// TIA Portal V20 export
// export: Created 2026-04-11T06:02:30.246913Z, ExportSetting WithDefaults, DisplayName Totally Integrated Automation Portal, DisplayVersion V20, DisplayName TIA Portal Openness, DisplayVersion V20, DisplayName TIA Portal Version Control Interface, DisplayVersion V20, DisplayName STEP 7 Professional, DisplayVersion V20, DisplayName STEP 7 Safety, DisplayVersion V20, DisplayName WinCC Basic/Comfort/Advanced, DisplayVersion V20, DisplayName WinCC Unified, DisplayVersion V20
TYPE "udtHMI_AnalogOutput"
// stored: IsFailsafeCompliant false
   STRUCT
      iMode : Int;   // Current mode
      iErrorCode { ExternalWritable := 'False'} : Int;   // Error code
      rValue { ExternalWritable := 'False'} : Real;   // Output Value
      rAutoValue { ExternalWritable := 'False'} : Real;   // Auto mode value
      rManualValue { S7_SetPoint := 'True'} : Real;   // Manual mode value
      rEstopValue { S7_SetPoint := 'True'} : Real;   // Estop condition custom value
      bPB_ResetError : Bool;   // PB Reset block errors
      bPBEN_ResetError { ExternalWritable := 'False'} : Bool;   // PB Reset error enabled
      bError { ExternalWritable := 'False'} : Bool;   // Overall error
      bInterlock { ExternalWritable := 'False'} : Bool;   // Analog output is interlocked
      iEstopFunction { S7_SetPoint := 'True'} : Int;   // Enum of E-Stop repsonse (Estop.xxx)
   END_STRUCT;
END_TYPE
